KUKA KRL program: test.src

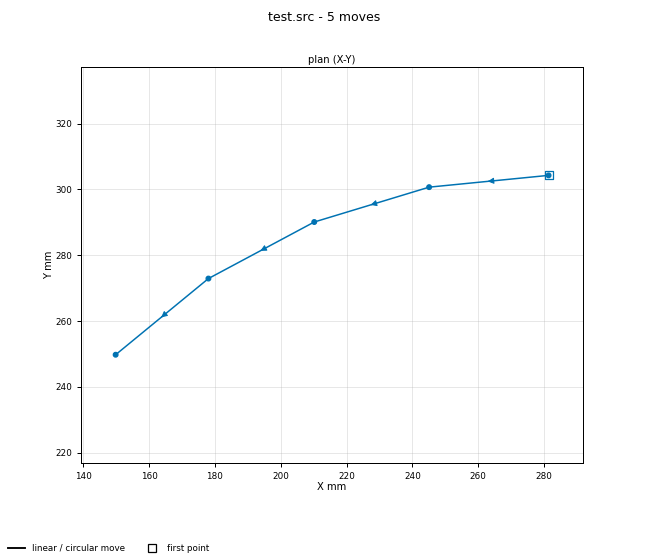
[picture p0: tool path of test.src, 5 of 7 moves have a stored position in this frame; points joined in program order, loops and branches not executed]
&ACCESS RVP
&REL 1
&PARAM TEMPLATE = C:\KRC\Roboter\Template\vorgabe
&PARAM EDITMASK = *
DEF test()

;FOLD INI
;FOLD BASISTECH INI
GLOBAL INTERRUPT DECL 3 WHEN $STOPMESS==TRUE DO IR_STOPM()
INTERRUPT ON 3
BAS(#INITMOV, 0)
;ENDFOLD (BASISTECH INI)
;ENDFOLD (INI)

;FOLD STARTPOSITION - BASE IS 1, TOOL IS 1, SPEED IS 15%, POSITION IS A1 5, A2 -90, A3 100, A4 5, A5 -10, A6 -5, E1 0, E2 0, E3 0, E4 0
$BWDSTART = FALSE
PDAT_ACT = {VEL 15, ACC 100, APO_DIST 50}
FDAT_ACT = {TOOL_NO 1, BASE_NO 1, IPO_FRAME #BASE}
BAS(#PTP_PARAMS, 15)
;ENDFOLD

;FOLD LIN SPEED IS 0.05 m/sec, INTERPOLATION SETTINGS IN FOLD
$VEL.CP=0.05
$ADVANCE=3
;ENDFOLD
PTP {A1 5, A2 -90, A3 100, A4 5, A5 -10, A6 -5, E1 0, E2 0, E3 0, E4 0}
$OUT[2] = TRUE
PTP {X 281.36, Y 304.25, Z 459.51, A 0, B 90, C 0}
LIN {X 245.07, Y 300.67, Z 459.51, A 0, B 90, C 0} C_DIS
LIN {X 210.17, Y 290.08, Z 459.51, A 0, B 90, C 0} C_DIS
LIN {X 178.02, Y 272.9, Z 459.51, A 0, B 90, C 0} C_DIS
LIN {X 149.83, Y 249.76, Z 459.51, A 0, B 90, C 0} C_DIS
$OUT[2] = FALSE
PTP {A1 5, A2 -90, A3 100, A4 5, A5 -10, A6 -5, E1 0, E2 0, E3 0, E4 0} C_PTP
;ENDFOLD

END
